TYPE
    ST_PlateInfo : STRUCT
        BoardID         : STRING;
        PlateID         : STRING;
        PlateNumber     : INT;
        PlateDimensions : STRING; // Dimension information of the plate (length, width, gauge)
        PlateGauge      : STRING;
        PlateWidth      : REAL;
        PlateHeight     : REAL;
        PlatePlaceX     : REAL;
        PlatePlaceY     : REAL;
        PlatePlaceAngle : REAL;
        TopOrBottom     : STRING; // Indicates if plate is on top or bottom of the board
    END_STRUCT
END_TYPE

(* stored: Version 1.1.0.1
   DUT ST_PlateInfo: Id {62b93293-007b-4d1c-a51a-19431f2f62e3} *)
